FUNCTION_BLOCK pH_control
  (* Standard: 61499-2 *)
  (* Version 0.1, 2015-00-21, Th?o, PC_THEO *)
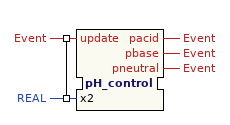
  EVENT_INPUT
    update WITH x2;
  END_EVENT
  EVENT_OUTPUT
    pacid;
    pbase;
    pneutral;
  END_EVENT
  VAR_INPUT
    x2 : REAL;
  END_VAR
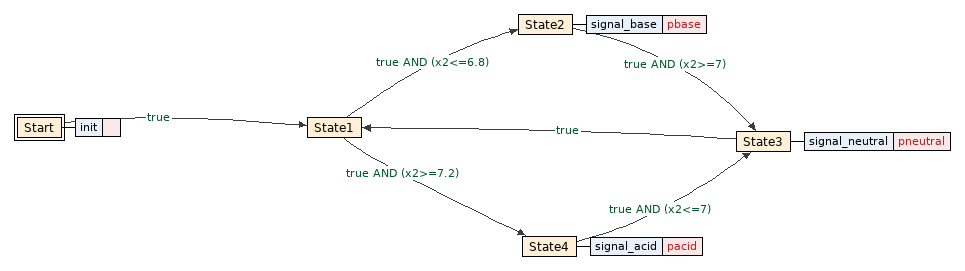
  EC_STATES
    Start : init;
    State1;
    State2 : signal_base -> pbase;
    State3 : signal_neutral -> pneutral;
    State4 : signal_acid -> pacid;
  END_STATES
  EC_TRANSITIONS
    Start TO State1 := true;
    State1 TO State2 := true AND (x2<=6.8);
    State1 TO State4 := true AND (x2>=7.2);
    State2 TO State3 := true AND (x2>=7);
    State3 TO State1 := true;
    State4 TO State3 := true AND (x2<=7);
  END_TRANSITIONS
  ALGORITHM init IN C:
me->x2=7.1;
  END_ALGORITHM
  ALGORITHM signal_base IN C:
printf("Send signal: pour base. Current pH: %f\n", me->x2);
  END_ALGORITHM
  ALGORITHM signal_neutral IN C:
printf("Send signal: pour neutral. Current pH: %f\n", me->x2);
  END_ALGORITHM
  ALGORITHM signal_acid IN C:
printf("Send signal: pour acid. Current pH: %f\n", me->x2);
  END_ALGORITHM
END_FUNCTION_BLOCK
